// TwinCAT 3 PLC project Provider
// ProgramVersion: 3.1.4023.0
// libraries:
//   Tc2_Standard, * (Beckhoff Automation GmbH)
//   Tc2_System, * (Beckhoff Automation GmbH)
//   Tc3_Module, * (Beckhoff Automation GmbH)
// project tree:
//   / PlcTask.TcTTO
//   POUs/ FB_Math.TcPOU, MAIN.TcPOU
// real-time tasks:
//   TASK PlcTask: cycle T#10ms, priority 20, ADS port 350
//   TASK PlcTask1: cycle T#10ms, priority 21, ADS port 351

CONFIGURATION Provider
    RESOURCE PLC ON TwinCAT3
        TASK PlcTask(INTERVAL := T#10ms, PRIORITY := 20);
        PROGRAM MAIN WITH PlcTask : MAIN;
    END_RESOURCE
END_CONFIGURATION

// ---- POUs/MAIN.TcPOU
PROGRAM MAIN
VAR
	fbMath	:FB_Math;
	icnt	:UDINT;
END_VAR

icnt:=icnt+1;

END_PROGRAM

// ---- POUs/FB_Math.TcPOU
FUNCTION_BLOCK FB_Math
VAR_INPUT
END_VAR
VAR_OUTPUT
END_VAR
VAR
END_VAR

{attribute'TcRpcEnable'}
METHOD M_ADD 	: LREAL
VAR_INPUT
	Param		:M_ADD_Parameters;
END_VAR
VAR_INST
	LastResult	:LREAL;
END_VAR
M_ADD		:=Param.A+Param.B;
LastResult	:=M_ADD;
END_METHOD

END_FUNCTION_BLOCK
